// TIA Portal V17 export
// export: Created 2025-03-07T09:23:49.3600816Z, ExportSetting WithDefaults, DisplayName Totally Integrated Automation Portal, DisplayVersion V17 Update 8, DisplayName TIA Portal Openness, DisplayVersion V17 Update 8, DisplayName TIA Portal Version Control Interface, DisplayVersion V17, DisplayName SINAMICS Startdrive Advanced, DisplayVersion V17 SP2, DisplayName SINAMICS Startdrive G110M, G120, G120C, G120D, G120P, G115D, DisplayVersion V17 SP2, DisplayName SINAMICS Startdrive G130, G150, S120, S150, SINAMICS MV, S210, DisplayVersion V17 SP2, DisplayName STEP 7 Professional, DisplayVersion V17 Update 8, DisplayName SINUMERIK ONE STEP 7 Toolbox, DisplayVersion V17 Update 12, DisplayName SINUMERIK 840D sl STEP 7 Toolbox, DisplayVersion V17 Update 12, DisplayName STEP 7 Safety, DisplayVersion V17 Update 6, DisplayName WinCC Advanced, DisplayVersion V17 Update 8
DATA_BLOCK "DB2050_HARDWARE_SOFTWARE_ENABLE_DISABLE"   // DB2050
{ S7_Optimized_Access := 'FALSE'; DB_Accessible_From_OPC_UA := 'FALSE' }
AUTHOR : ETXETAR
VERSION : 1.0
// stored: AutoNumber false, DBAccessibleFromOPCUA false, DBAccessibleFromWebserver true, IsOnlyStoredInLoadMemory false, IsWriteProtectedInAS false
   VAR RETAIN
      DISABLE_PART : Struct
         HW_GENERAL_CONDITIONS : Bool;   // HARDWARE GENERAL CONDITIONS
         SW_GENERAL_CONDITIONS : Bool;   // SOFTWARE GENERAL CONDITIONS
         PART_A_ENABLE : Bool;   // PART A ENABLE
         PART_B_ENABLE : Bool;   // PART B ENABLE
         PART_C_ENABLE : Bool;   // PART C ENABLE
         PART_D_ENABLE : Bool;   // PART D ENABLE
         PART_E_ENABLE : Bool;   // PART E ENABLE
         PART_F_ENABLE : Bool;   // PART F ENABLE
         HW_PART_A_ENABLE_REQUEST : Bool;   // HARDWARE PART A ENABLE REQUEST
         HW_PART_A_DISABLE_REQUEST : Bool;   // HARDWARE PART A DISABLE REQUEST
         HW_PART_B_ENABLE_REQUEST : Bool;   // HARDWARE PART B ENABLE REQUEST
         HW_PART_B_DISABLE_REQUEST : Bool;   // HARDWARE PART B DISABLE REQUEST
         HW_PART_C_ENABLE_REQUEST : Bool;   // HARDWARE PART C ENABLE REQUEST
         HW_PART_C_DISABLE_REQUEST : Bool;   // HARDWARE PART C DISABLE REQUEST
         HW_PART_D_ENABLE_REQUEST : Bool;   // HARDWARE PART D ENABLE REQUEST
         HW_PART_D_DISABLE_REQUEST : Bool;   // HARDWARE PART D DISABLE REQUEST
         HW_PART_E_ENABLE_REQUEST : Bool;   // HARDWARE PART E ENABLE REQUEST
         HW_PART_E_DISABLE_REQUEST : Bool;   // HARDWARE PART E DISABLE REQUEST
         HW_PART_F_ENABLE_REQUEST : Bool;   // HARDWARE PART F ENABLE REQUEST
         HW_PART_F_DISABLE_REQUEST : Bool;   // HARDWARE PART F DISABLE REQUEST
         HW_PART_ENABLE_DISABLE_REQUEST : Bool;   // HARDWARE ENABLE DISABLE REQUEST
         SW_PART_A_ENABLE_REQUEST : Bool;   // SOFTWARE PART A ENABLE REQUEST
         SW_PART_A_DISABLE_REQUEST : Bool;   // SOFTWARE PART A DISABLE REQUEST
         SW_PART_B_ENABLE_REQUEST : Bool;   // SOFTWARE PART B ENABLE REQUEST
         SW_PART_B_DISABLE_REQUEST : Bool;   // SOFTWARE PART B DISABLE REQUEST
         SW_PART_C_ENABLE_REQUEST : Bool;   // SOFTWARE PART C ENABLE REQUEST
         SW_PART_C_DISABLE_REQUEST : Bool;   // SOFTWARE PART C DISABLE REQUEST
         SW_PART_D_ENABLE_REQUEST : Bool;   // SOFTWARE PART D ENABLE REQUEST
         SW_PART_D_DISABLE_REQUEST : Bool;   // SOFTWARE PART D DISABLE REQUEST
         SW_PART_E_ENABLE_REQUEST : Bool;   // SOFTWARE PART E ENABLE REQUEST
         SW_PART_E_DISABLE_REQUEST : Bool;   // SOFTWARE PART E DISABLE REQUEST
         SW_PART_F_ENABLE_REQUEST : Bool;   // SOFTWARE PART F ENABLE REQUEST
         SW_PART_F_DISABLE_REQUEST : Bool;   // SOFTWARE PART F DISABLE REQUEST
         SW_PART_ENABLE_DISABLE_REQUEST : Bool;   // SOFTWARE ENABLE DISABLE REQUEST
         HMI_ACCEPT_BUTTON : Bool;   // HMI ACCEPT BUTTON
         HW_PART_A_ENABLED : Bool := true;   // HARDWARE PART A ENABLED
         HW_PART_B_ENABLED : Bool := true;   // HARDWARE PART B ENABLED
         HW_PART_C_ENABLED : Bool := true;   // HARDWARE PART C ENABLED
         HW_PART_D_ENABLED : Bool;   // HARDWARE PART D ENABLED
         HW_PART_E_ENABLED : Bool;   // HARDWARE PART E ENABLED
         HW_PART_F_ENABLED : Bool;   // HARDWARE PART F ENABLED
         SW_PART_A_ENABLED : Bool := true;   // SOFTWARE PART A ENABLED
         SW_PART_B_ENABLED : Bool := true;   // SOFTWARE PART B ENABLED
         SW_PART_C_ENABLED : Bool := true;   // SOFTWARE PART C ENABLED
         SW_PART_D_ENABLED : Bool;   // SOFTWARE PART D ENABLED
         SW_PART_E_ENABLED : Bool;   // SOFTWARE PART E ENABLED
         SW_PART_F_ENABLED : Bool;   // SOFTWARE PART F ENABLED
         PART_A_DISABLE_ALARM : Bool;   // PART A DISABLE ALARM
         PART_B_DISABLE_ALARM : Bool;   // PART B DISABLE ALARM
         PART_C_DISABLE_ALARM : Bool;   // PART C DISABLE ALARM
         PART_D_DISABLE_ALARM : Bool;   // PART D DISABLE ALARM
         PART_E_DISABLE_ALARM : Bool;   // PART E DISABLE ALARM
         PART_F_DISABLE_ALARM : Bool;   // PART F DISABLE ALARM
         DESELECT_IN_PROGRESS : Bool;   // DESELECTION IN PROGRESS
         HW_DISABLED_ACK : Bool;   // HARDWARE DISABLED ACKNOWLEDGE
         HW_DISABLED_ACK_AUX : Bool;   // HARDWARE DISABLED ACKNOWLEDGE AUXILIARY
         ALL_HW_PARTS_DISABLED : Bool;   // ALL HARDWARE PARTS DISABLED
         ALL_SW_PARTS_DISABLED : Bool;   // ALL SOFTWARE PARTS DISABLED
         ALL_HARDWARE_ENABLED : Bool;   // ALL HARDWARE ENABLED
         PART_A_DISABLED_SCRIPT_COMMAND : Bool;   // PART A DISABLED SCRIPT COMMAND
         PART_A_ENABLED_SCRIPT_COMMAND : Bool;   // PART A ENABLED SCRIPT COMMAND
         PART_B_DISABLED_SCRIPT_COMMAND : Bool;   // PART B DISABLED SCRIPT COMMAND
         PART_B_ENABLED_SCRIPT_COMMAND : Bool;   // PART B ENABLED SCRIPT COMMAND
         PART_C_DISABLED_SCRIPT_COMMAND : Bool;   // PART C DISABLED SCRIPT COMMAND
         PART_C_ENABLED_SCRIPT_COMMAND : Bool;   // PART C ENABLED SCRIPT COMMAND
         PART_D_DISABLED_SCRIPT_COMMAND : Bool;   // PART D DISABLED SCRIPT COMMAND
         PART_D_ENABLED_SCRIPT_COMMAND : Bool;   // PART D ENABLED SCRIPT COMMAND
         PART_E_DISABLED_SCRIPT_COMMAND : Bool;   // PART E DISABLED SCRIPT COMMAND
         PART_E_ENABLED_SCRIPT_COMMAND : Bool;   // PART E ENABLED SCRIPT COMMAND
         PART_F_DISABLED_SCRIPT_COMMAND : Bool;   // PART F DISABLED SCRIPT COMMAND
         PART_F_ENABLED_SCRIPT_COMMAND : Bool;   // PART F ENABLED SCRIPT COMMAND
         ALARM_SCREEN : Int;   // HMI ALARMS SCREEN NUMBER
         ENABLE_MACHINE_STRUCTURE_SCREEN : Int;   // HMI ENABLE MACHINE STRUCTURE SCREEN NUMBER
         SW_PULSE : Array[1..16] of Bool;
         HW_PULSE : Array[1..16] of Bool;
      END_STRUCT;
   END_VAR
BEGIN
END_DATA_BLOCK
